FUNCTION_BLOCK FB_SerialCom
VAR_IN_OUT
	TxBuffer			: ComBuffer;
	RxBuffer			: ComBuffer;
END_VAR
VAR
	fbReceive			: ReceiveString;
	sReceivedString		: STRING;
	bStringReceived		: BOOL;
	bReceiveBusy		: BOOL;
	bReceiveError		: BOOL;
	eReceiveErrorID		: ComError_t;
	bReceiveTimeout		: BOOL;
END_VAR
VAR_OUTPUT
	sHeidOut 			: STRING;
	Error				: BOOL := FALSE;
END_VAR

//	Receive string data:
//	The block receives any data strings beginning with a STX ($02) and ending with an ETX ($03) character.	
fbReceive(
	Prefix:= '',
	Suffix:= '',
	Timeout:= T#1s,
	ReceivedString := sHeidOut,
	RXbuffer:= RxBuffer,
	StringReceived=> bStringReceived,
	Busy => bReceiveBusy,
	Error => ,
	RxTimeout => bReceiveTimeout );
IF fbReceive.Error <> COMERROR_NOERROR THEN
	eReceiveErrorID := fbReceive.Error;
	//Error := TRUE;
END_IF

END_FUNCTION_BLOCK

(* stored: Version 1.1.0.1, ProductVersion 3.1.4024.2
   POU FB_SerialCom: Id {181e7c70-138b-446a-a6f5-34e588388885}, SpecialFunc None *)
